Fanuc KAREL source: ADD_STRINGPC.kl

PROGRAM T
%NOLOCKGROUP
VAR
 v0 : ARRAY[20] OF BYTE
 v1 : INTEGER
 v2 : STRING[40]
 v3 : INTEGER
BEGIN
 ADD_STRINGPC(v0, v1, v2, v3)
END T
